Yaskawa INFORM job: linear.JBI

/JOB
//NAME AAA
//POS
///NPOS 2,0,0,0,0,0
C00000=-48629,112084,69901,4161,-52375,-4796
C00001=-46969,105372,61036,4871,-50464,-5567
//INST
///DATE 2023/02/07 09:03
///ATTR SC,RW
///GROUP1 RB1
NOP
MOVL C00000 V=10.0 PL=8
MOVL C00001 V=10.0 PL=0
END
